KUKA KRL data list: $config.dat

&ACCESS RV$
&REL 2
DEFDAT  $CONFIG

INT COM_ACTION=2
INT COM_ACTCNT=0
REAL COM_ROUNDM=-1.00000
REAL COM_VALUE1=0.0
REAL COM_VALUE2=0.0
REAL COM_VALUE3=0.0
REAL COM_VALUE4=0.0
DECL E6AXIS COM_E6AXIS
DECL POS COM_POS
DECL FRAME COM_FRAME
DECL E6POS COM_E6POS

DECL REAL WAAM_VEL = 0.05    ; Default linear velocity for deposition in m/s
DECL REAL WAAM_ACC = 0.6     ; Default acceleration for deposition in m/s^2
DECL REAL WAAM_APPROACH_VEL = 50 ; Approach velocity in % for PTP movements
DECL POS WAAM_POS
ENDDAT
